FUNCTION_BLOCK FB_MoveVelocity
VAR_INPUT
	fTargetVelocity 	: REAL;
	fAccMax 			: REAL;
	fDecMax 			: REAL;
END_VAR

VAR
	_fVelocity 			: REAL;	
	_fAcc 				: REAL;
	_bIsReached			: BOOL;
	fVelocityTolerance	: REAL;
END_VAR

_bIsReached := FALSE;
IF _fAcc = 0 THEN
	IF ABS(fAccMax) > ABS(fDecMax) THEN
		fVelocityTolerance := ABS(fAccMax) * GVL_Core.fbSystem.fDeltaTime * GVL_Core.fbSystem.fTimeScaling;
	ELSE
		fVelocityTolerance := ABS(fDecMax) * GVL_Core.fbSystem.fDeltaTime * GVL_Core.fbSystem.fTimeScaling;
	END_IF
ELSE
	fVelocityTolerance := ABS(_fAcc) * GVL_Core.fbSystem.fDeltaTime * GVL_Core.fbSystem.fTimeScaling;
END_IF	

(* Calculate acceleration *)
//Hold velocity (velocity reached)
IF F_Compare(fVelocity, fTargetVelocity, fVelocityTolerance) THEN
	_fAcc := 0;
	_fVelocity := fTargetVelocity;
	_bIsReached := TRUE;
	RETURN;
END_IF

IF _fVelocity - fTargetVelocity > fVelocityTolerance THEN
	//Decelerate
	IF _fVelocity < 0 THEN
		_fAcc := -ABS(fAccMax);
	ELSE
		_fAcc := -ABS(fDecMax);
	END_IF
 ELSIF _fVelocity - fTargetVelocity < -fVelocityTolerance THEN
	//Accelerate
	IF _fVelocity < 0 THEN
		_fAcc := ABS(fDecMax);
	ELSE
		_fAcc := ABS(fAccMax);
	END_IF
END_IF

_fVelocity := _fVelocity + _fAcc * GVL_Core.fbSystem.fDeltaTime * GVL_Core.fbSystem.fTimeScaling;
_bIsReached := F_Compare(_fVelocity, fTargetVelocity, fVelocityTolerance);

PROPERTY bIsReached : BOOL
GET
bIsReached := THIS^._bIsReached;
END_GET
END_PROPERTY

PROPERTY fAcc : REAL
GET
fAcc := THIS^._fAcc;
END_GET
SET
THIS^._fAcc := fAcc;
END_SET
END_PROPERTY

PROPERTY fVelocity : REAL
GET
fVelocity := THIS^._fVelocity;
END_GET
SET
THIS^._fVelocity := fVelocity;
END_SET
END_PROPERTY

END_FUNCTION_BLOCK

(* stored: Version 1.1.0.1, ProductVersion 3.1.4024.12
   POU FB_MoveVelocity: Id {9bae960a-d9ba-07f3-39f8-a131e14eb6c6}, SpecialFunc None
   Property bIsReached: Id {1b62f692-0ce8-0ddf-04df-a2cb5441658f}
   Get Get: Id {f53b033e-df5e-07b6-2792-bf6722784217}
   Property fAcc: Id {d6f7d3ff-b9bd-097a-2fcb-bea90667f161}
   Get Get: Id {e64a8ff4-07d9-014d-1950-84da0b2118c2}
   Set Set: Id {d4288bbd-43fe-05dc-3465-dbb413486a26}
   Property fVelocity: Id {ba9df249-e9e4-070c-3e5e-4885a73cc59a}
   Get Get: Id {85b8344d-47b3-05d3-3895-9954bbfd24d7}
   Set Set: Id {ea155c37-d5a6-046b-2346-08eea0da3f92} *)
